// TIA Portal V20 export
TYPE "LER_typePartDataEm7"
// stored: Access Published
   STRUCT
      sepaGripper : "LER_typeCommonData";
      winder : "LER_typeCommonData";
   END_STRUCT;
END_TYPE
